// NeuroPLC ¡ª FourierKAN [28,16,4]
// C^2-BV Architecture: FourierKAN compiled via universal LUT extraction
// LUT points: 15, domain: [-3.0, 3.0]
// Proposition 9: M2 bounds guaranteed by C^2 property

FUNCTION_BLOCK "NeuroPLC_FourierKAN"
VAR_INPUT
    "feat_1" : REAL;
    "feat_2" : REAL;
    "feat_3" : REAL;
    "feat_4" : REAL;
    "feat_5" : REAL;
    "feat_6" : REAL;
    "feat_7" : REAL;
    "feat_8" : REAL;
    "feat_9" : REAL;
    "feat_10" : REAL;
    "feat_11" : REAL;
    "feat_12" : REAL;
    "feat_13" : REAL;
    "feat_14" : REAL;
    "feat_15" : REAL;
    "feat_16" : REAL;
    "feat_17" : REAL;
    "feat_18" : REAL;
    "feat_19" : REAL;
    "feat_20" : REAL;
    "feat_21" : REAL;
    "feat_22" : REAL;
    "feat_23" : REAL;
    "feat_24" : REAL;
    "feat_25" : REAL;
    "feat_26" : REAL;
    "feat_27" : REAL;
    "feat_28" : REAL;
    "trigger" : BOOL;
END_VAR

VAR_OUTPUT
    "class_output_1" : REAL;
    "class_output_2" : REAL;
    "class_output_3" : REAL;
    "class_output_4" : REAL;
    "max_confidence" : REAL;
    "predicted_class" : INT;
END_VAR

VAR
    "layer0_out_1" : REAL := 0.0;
    "layer0_out_2" : REAL := 0.0;
    "layer0_out_3" : REAL := 0.0;
    "layer0_out_4" : REAL := 0.0;
    "layer0_out_5" : REAL := 0.0;
    "layer0_out_6" : REAL := 0.0;
    "layer0_out_7" : REAL := 0.0;
    "layer0_out_8" : REAL := 0.0;
    "layer0_out_9" : REAL := 0.0;
    "layer0_out_10" : REAL := 0.0;
    "layer0_out_11" : REAL := 0.0;
    "layer0_out_12" : REAL := 0.0;
    "layer0_out_13" : REAL := 0.0;
    "layer0_out_14" : REAL := 0.0;
    "layer0_out_15" : REAL := 0.0;
    "layer0_out_16" : REAL := 0.0;
    "layer1_out_1" : REAL := 0.0;
    "layer1_out_2" : REAL := 0.0;
    "layer1_out_3" : REAL := 0.0;
    "layer1_out_4" : REAL := 0.0;
    "i" : INT;
    "k" : INT;
    "t" : REAL;
    "max_val" : REAL;
    "max_idx" : INT;
END_VAR

BEGIN
    IF NOT "trigger" THEN RETURN; END_IF;

    // === Layer 0 (28 -> 16) ===
    "layer0_out_1" := 0.0;
    // Edge (1->1): LUT interpolation
    "k" := 1;
    FOR "i" := 2 TO 15 DO
        IF "feat_1" >= -3.000000 AND "feat_1" <= 3.000000 THEN
    END_FOR;
    // Edge (2->1): LUT interpolation
    "k" := 1;
    FOR "i" := 2 TO 15 DO
    END_FOR;
    // Edge (3->1): LUT interpolation
    "k" := 1;
    FOR "i" := 2 TO 15 DO
    END_FOR;
    // Edge (4->1): LUT interpolation
    "k" := 1;
    FOR "i" := 2 TO 15 DO
    END_FOR;
    // Edge (5->1): LUT interpolation
    "k" := 1;
    FOR "i" := 2 TO 15 DO
    END_FOR;
    // Edge (6->1): LUT interpolation
    "k" := 1;
    FOR "i" := 2 TO 15 DO
    END_FOR;
    // Edge (7->1): LUT interpolation
    "k" := 1;
    FOR "i" := 2 TO 15 DO
    END_FOR;
    // Edge (8->1): LUT interpolation
    "k" := 1;
    FOR "i" := 2 TO 15 DO
    END_FOR;
    // Edge (9->1): LUT interpolation
    "k" := 1;
    FOR "i" := 2 TO 15 DO
    END_FOR;
    // Edge (10->1): LUT interpolation
    "k" := 1;
    FOR "i" := 2 TO 15 DO
    END_FOR;
    // Edge (11->1): LUT interpolation
    "k" := 1;
    FOR "i" := 2 TO 15 DO
    END_FOR;
    // Edge (12->1): LUT interpolation
    "k" := 1;
    FOR "i" := 2 TO 15 DO
    END_FOR;
    // Edge (13->1): LUT interpolation
    "k" := 1;
    FOR "i" := 2 TO 15 DO
    END_FOR;
    // Edge (14->1): LUT interpolation
    "k" := 1;
    FOR "i" := 2 TO 15 DO
    END_FOR;
    // Edge (15->1): LUT interpolation
    "k" := 1;
    FOR "i" := 2 TO 15 DO
    END_FOR;
    // Edge (16->1): LUT interpolation
    "k" := 1;
    FOR "i" := 2 TO 15 DO
    END_FOR;
    // Edge (17->1): LUT interpolation
    "k" := 1;
    FOR "i" := 2 TO 15 DO
    END_FOR;
    // Edge (18->1): LUT interpolation
    "k" := 1;
    FOR "i" := 2 TO 15 DO
    END_FOR;
    // Edge (19->1): LUT interpolation
    "k" := 1;
    FOR "i" := 2 TO 15 DO
    END_FOR;
    // Edge (20->1): LUT interpolation
    "k" := 1;
    FOR "i" := 2 TO 15 DO
    END_FOR;
    // Edge (21->1): LUT interpolation
    "k" := 1;
    FOR "i" := 2 TO 15 DO
    END_FOR;
    // Edge (22->1): LUT interpolation
    "k" := 1;
    FOR "i" := 2 TO 15 DO
    END_FOR;
    // Edge (23->1): LUT interpolation
    "k" := 1;
    FOR "i" := 2 TO 15 DO
    END_FOR;
    // Edge (24->1): LUT interpolation
    "k" := 1;
    FOR "i" := 2 TO 15 DO
    END_FOR;
    // Edge (25->1): LUT interpolation
    "k" := 1;
    FOR "i" := 2 TO 15 DO
    END_FOR;
    // Edge (26->1): LUT interpolation
    "k" := 1;
    FOR "i" := 2 TO 15 DO
    END_FOR;
    // Edge (27->1): LUT interpolation
    "k" := 1;
    FOR "i" := 2 TO 15 DO
    END_FOR;
    // Edge (28->1): LUT interpolation
    "k" := 1;
    FOR "i" := 2 TO 15 DO
    END_FOR;
    "layer0_out_2" := 0.0;
    // Edge (1->2): LUT interpolation
    "k" := 1;
    FOR "i" := 2 TO 15 DO
    END_FOR;
    // Edge (2->2): LUT interpolation
    "k" := 1;
    FOR "i" := 2 TO 15 DO
    END_FOR;
    // Edge (3->2): LUT interpolation
    "k" := 1;
    FOR "i" := 2 TO 15 DO
    END_FOR;
    // Edge (4->2): LUT interpolation
    "k" := 1;
    FOR "i" := 2 TO 15 DO
    END_FOR;
    // Edge (5->2): LUT interpolation
    "k" := 1;
    FOR "i" := 2 TO 15 DO
    END_FOR;
    // Edge (6->2): LUT interpolation
    "k" := 1;
    FOR "i" := 2 TO 15 DO
    END_FOR;
    // Edge (7->2): LUT interpolation
    "k" := 1;
    FOR "i" := 2 TO 15 DO
    END_FOR;
    // Edge (8->2): LUT interpolation
    "k" := 1;
    FOR "i" := 2 TO 15 DO
    END_FOR;
    // Edge (9->2): LUT interpolation
    "k" := 1;
    FOR "i" := 2 TO 15 DO
    END_FOR;
    // Edge (10->2): LUT interpolation
    "k" := 1;
    FOR "i" := 2 TO 15 DO
    END_FOR;
    // Edge (11->2): LUT interpolation
    "k" := 1;
    FOR "i" := 2 TO 15 DO
    END_FOR;
    // Edge (12->2): LUT interpolation
    "k" := 1;
    FOR "i" := 2 TO 15 DO
    END_FOR;
    // Edge (13->2): LUT interpolation
    "k" := 1;
    FOR "i" := 2 TO 15 DO
    END_FOR;
    // Edge (14->2): LUT interpolation
    "k" := 1;
    FOR "i" := 2 TO 15 DO
    END_FOR;
    // Edge (15->2): LUT interpolation
    "k" := 1;
    FOR "i" := 2 TO 15 DO
    END_FOR;
    // Edge (16->2): LUT interpolation
    "k" := 1;
    FOR "i" := 2 TO 15 DO
    END_FOR;
    // Edge (17->2): LUT interpolation
    "k" := 1;
    FOR "i" := 2 TO 15 DO
    END_FOR;
    // Edge (18->2): LUT interpolation
    "k" := 1;
    FOR "i" := 2 TO 15 DO
    END_FOR;
    // Edge (19->2): LUT interpolation
    "k" := 1;
    FOR "i" := 2 TO 15 DO
    END_FOR;
    // Edge (20->2): LUT interpolation
    "k" := 1;
    FOR "i" := 2 TO 15 DO
    END_FOR;
    // Edge (21->2): LUT interpolation
    "k" := 1;
    FOR "i" := 2 TO 15 DO
    END_FOR;
    // Edge (22->2): LUT interpolation
    "k" := 1;
    FOR "i" := 2 TO 15 DO
    END_FOR;
    // Edge (23->2): LUT interpolation
    "k" := 1;
    FOR "i" := 2 TO 15 DO
    END_FOR;
    // Edge (24->2): LUT interpolation
    "k" := 1;
    FOR "i" := 2 TO 15 DO
    END_FOR;
    // Edge (25->2): LUT interpolation
    "k" := 1;
    FOR "i" := 2 TO 15 DO
    END_FOR;
    // Edge (26->2): LUT interpolation
    "k" := 1;
    FOR "i" := 2 TO 15 DO
    END_FOR;
    // Edge (27->2): LUT interpolation
    "k" := 1;
    FOR "i" := 2 TO 15 DO
    END_FOR;
    // Edge (28->2): LUT interpolation
    "k" := 1;
    FOR "i" := 2 TO 15 DO
    END_FOR;
    "layer0_out_3" := 0.0;
    // Edge (1->3): LUT interpolation
    "k" := 1;
    FOR "i" := 2 TO 15 DO
    END_FOR;
    // Edge (2->3): LUT interpolation
    "k" := 1;
    FOR "i" := 2 TO 15 DO
    END_FOR;
    // Edge (3->3): LUT interpolation
    "k" := 1;
    FOR "i" := 2 TO 15 DO
    END_FOR;
    // Edge (4->3): LUT interpolation
    "k" := 1;
    FOR "i" := 2 TO 15 DO
    END_FOR;
    // Edge (5->3): LUT interpolation
    "k" := 1;
    FOR "i" := 2 TO 15 DO
    END_FOR;
    // Edge (6->3): LUT interpolation
    "k" := 1;
    FOR "i" := 2 TO 15 DO
    END_FOR;
    // Edge (7->3): LUT interpolation
    "k" := 1;
    FOR "i" := 2 TO 15 DO
    END_FOR;
    // Edge (8->3): LUT interpolation
    "k" := 1;
    FOR "i" := 2 TO 15 DO
    END_FOR;
    // Edge (9->3): LUT interpolation
    "k" := 1;
    FOR "i" := 2 TO 15 DO
    END_FOR;
    // Edge (10->3): LUT interpolation
    "k" := 1;
    FOR "i" := 2 TO 15 DO
    END_FOR;
    // Edge (11->3): LUT interpolation
    "k" := 1;
    FOR "i" := 2 TO 15 DO
    END_FOR;
    // Edge (12->3): LUT interpolation
    "k" := 1;
    FOR "i" := 2 TO 15 DO
    END_FOR;
    // Edge (13->3): LUT interpolation
    "k" := 1;
    FOR "i" := 2 TO 15 DO
    END_FOR;
    // Edge (14->3): LUT interpolation
    "k" := 1;
    FOR "i" := 2 TO 15 DO
    END_FOR;
    // Edge (15->3): LUT interpolation
    "k" := 1;
    FOR "i" := 2 TO 15 DO
    END_FOR;
    // Edge (16->3): LUT interpolation
    "k" := 1;
    FOR "i" := 2 TO 15 DO
    END_FOR;
    // Edge (17->3): LUT interpolation
    "k" := 1;
    FOR "i" := 2 TO 15 DO
    END_FOR;
    // Edge (18->3): LUT interpolation
    "k" := 1;
    FOR "i" := 2 TO 15 DO
    END_FOR;
    // Edge (19->3): LUT interpolation
    "k" := 1;
    FOR "i" := 2 TO 15 DO
    END_FOR;
    // Edge (20->3): LUT interpolation
    "k" := 1;
    FOR "i" := 2 TO 15 DO
    END_FOR;
    // Edge (21->3): LUT interpolation
    "k" := 1;
    FOR "i" := 2 TO 15 DO
    END_FOR;
    // Edge (22->3): LUT interpolation
    "k" := 1;
    FOR "i" := 2 TO 15 DO
    END_FOR;
    // Edge (23->3): LUT interpolation
    "k" := 1;
    FOR "i" := 2 TO 15 DO
    END_FOR;
    // Edge (24->3): LUT interpolation
    "k" := 1;
    FOR "i" := 2 TO 15 DO
    END_FOR;
    // Edge (25->3): LUT interpolation
    "k" := 1;
    FOR "i" := 2 TO 15 DO
    END_FOR;
    // Edge (26->3): LUT interpolation
    "k" := 1;
    FOR "i" := 2 TO 15 DO
    END_FOR;
    // Edge (27->3): LUT interpolation
    "k" := 1;
    FOR "i" := 2 TO 15 DO
    END_FOR;
    // Edge (28->3): LUT interpolation
    "k" := 1;
    FOR "i" := 2 TO 15 DO
    END_FOR;
    "layer0_out_4" := 0.0;
    // Edge (1->4): LUT interpolation
    "k" := 1;
    FOR "i" := 2 TO 15 DO
    END_FOR;
    // Edge (2->4): LUT interpolation
    "k" := 1;
    FOR "i" := 2 TO 15 DO
    END_FOR;
    // Edge (3->4): LUT interpolation
    "k" := 1;
    FOR "i" := 2 TO 15 DO
    END_FOR;
    // Edge (4->4): LUT interpolation
    "k" := 1;
    FOR "i" := 2 TO 15 DO
    END_FOR;
    // Edge (5->4): LUT interpolation
    "k" := 1;
    FOR "i" := 2 TO 15 DO
    END_FOR;
    // Edge (6->4): LUT interpolation
    "k" := 1;
    FOR "i" := 2 TO 15 DO
    END_FOR;
    // Edge (7->4): LUT interpolation
    "k" := 1;
    FOR "i" := 2 TO 15 DO
    END_FOR;
    // Edge (8->4): LUT interpolation
    "k" := 1;
    FOR "i" := 2 TO 15 DO
    END_FOR;
    // Edge (9->4): LUT interpolation
    "k" := 1;
    FOR "i" := 2 TO 15 DO
    END_FOR;
    // Edge (10->4): LUT interpolation
    "k" := 1;
    FOR "i" := 2 TO 15 DO
    END_FOR;
    // Edge (11->4): LUT interpolation
    "k" := 1;
    FOR "i" := 2 TO 15 DO
    END_FOR;
    // Edge (12->4): LUT interpolation
    "k" := 1;
    FOR "i" := 2 TO 15 DO
    END_FOR;
    // Edge (13->4): LUT interpolation
    "k" := 1;
    FOR "i" := 2 TO 15 DO
    END_FOR;
    // Edge (14->4): LUT interpolation
    "k" := 1;
    FOR "i" := 2 TO 15 DO
    END_FOR;
    // Edge (15->4): LUT interpolation
    "k" := 1;
    FOR "i" := 2 TO 15 DO
    END_FOR;
    // Edge (16->4): LUT interpolation
    "k" := 1;
    FOR "i" := 2 TO 15 DO
    END_FOR;
    // Edge (17->4): LUT interpolation
    "k" := 1;
    FOR "i" := 2 TO 15 DO
    END_FOR;
    // Edge (18->4): LUT interpolation
    "k" := 1;
    FOR "i" := 2 TO 15 DO
    END_FOR;
    // Edge (19->4): LUT interpolation
    "k" := 1;
    FOR "i" := 2 TO 15 DO
    END_FOR;
    // Edge (20->4): LUT interpolation
    "k" := 1;
    FOR "i" := 2 TO 15 DO
    END_FOR;
    // Edge (21->4): LUT interpolation
    "k" := 1;
    FOR "i" := 2 TO 15 DO
    END_FOR;
    // Edge (22->4): LUT interpolation
    "k" := 1;
    FOR "i" := 2 TO 15 DO
    END_FOR;
    // Edge (23->4): LUT interpolation
    "k" := 1;
    FOR "i" := 2 TO 15 DO
    END_FOR;
    // Edge (24->4): LUT interpolation
    "k" := 1;
    FOR "i" := 2 TO 15 DO
    END_FOR;
    // Edge (25->4): LUT interpolation
    "k" := 1;
    FOR "i" := 2 TO 15 DO
    END_FOR;
    // Edge (26->4): LUT interpolation
    "k" := 1;
    FOR "i" := 2 TO 15 DO
    END_FOR;
    // Edge (27->4): LUT interpolation
    "k" := 1;
    FOR "i" := 2 TO 15 DO
    END_FOR;
    // Edge (28->4): LUT interpolation
    "k" := 1;
    FOR "i" := 2 TO 15 DO
    END_FOR;
    "layer0_out_5" := 0.0;
    // Edge (1->5): LUT interpolation
    "k" := 1;
    FOR "i" := 2 TO 15 DO
    END_FOR;
    // Edge (2->5): LUT interpolation
    "k" := 1;
    FOR "i" := 2 TO 15 DO
    END_FOR;
    // Edge (3->5): LUT interpolation
    "k" := 1;
    FOR "i" := 2 TO 15 DO
    END_FOR;
    // Edge (4->5): LUT interpolation
    "k" := 1;
    FOR "i" := 2 TO 15 DO
    END_FOR;
    // Edge (5->5): LUT interpolation
    "k" := 1;
    FOR "i" := 2 TO 15 DO
    END_FOR;
    // Edge (6->5): LUT interpolation
    "k" := 1;
    FOR "i" := 2 TO 15 DO
    END_FOR;
    // Edge (7->5): LUT interpolation
    "k" := 1;
    FOR "i" := 2 TO 15 DO
    END_FOR;
    // Edge (8->5): LUT interpolation
    "k" := 1;
    FOR "i" := 2 TO 15 DO
    END_FOR;
    // Edge (9->5): LUT interpolation
    "k" := 1;
    FOR "i" := 2 TO 15 DO
    END_FOR;
    // Edge (10->5): LUT interpolation
    "k" := 1;
    FOR "i" := 2 TO 15 DO
    END_FOR;
    // Edge (11->5): LUT interpolation
    "k" := 1;
    FOR "i" := 2 TO 15 DO
    END_FOR;
    // Edge (12->5): LUT interpolation
    "k" := 1;
    FOR "i" := 2 TO 15 DO
    END_FOR;
    // Edge (13->5): LUT interpolation
    "k" := 1;
    FOR "i" := 2 TO 15 DO
    END_FOR;
    // Edge (14->5): LUT interpolation
    "k" := 1;
    FOR "i" := 2 TO 15 DO
    END_FOR;
    // Edge (15->5): LUT interpolation
    "k" := 1;
    FOR "i" := 2 TO 15 DO
    END_FOR;
    // Edge (16->5): LUT interpolation
    "k" := 1;
    FOR "i" := 2 TO 15 DO
    END_FOR;
    // Edge (17->5): LUT interpolation
    "k" := 1;
    FOR "i" := 2 TO 15 DO
    END_FOR;
    // Edge (18->5): LUT interpolation
    "k" := 1;
    FOR "i" := 2 TO 15 DO
    END_FOR;
    // Edge (19->5): LUT interpolation
    "k" := 1;
    FOR "i" := 2 TO 15 DO
    END_FOR;
    // Edge (20->5): LUT interpolation
    "k" := 1;
    FOR "i" := 2 TO 15 DO
    END_FOR;
    // Edge (21->5): LUT interpolation
    "k" := 1;
    FOR "i" := 2 TO 15 DO
    END_FOR;
    // Edge (22->5): LUT interpolation
    "k" := 1;
    FOR "i" := 2 TO 15 DO
    END_FOR;
    // Edge (23->5): LUT interpolation
    "k" := 1;
    FOR "i" := 2 TO 15 DO
    END_FOR;
    // Edge (24->5): LUT interpolation
    "k" := 1;
    FOR "i" := 2 TO 15 DO
    END_FOR;
    // Edge (25->5): LUT interpolation
    "k" := 1;
    FOR "i" := 2 TO 15 DO
    END_FOR;
    // Edge (26->5): LUT interpolation
    "k" := 1;
    FOR "i" := 2 TO 15 DO
    END_FOR;
    // Edge (27->5): LUT interpolation
    "k" := 1;
    FOR "i" := 2 TO 15 DO
    END_FOR;
    // Edge (28->5): LUT interpolation
    "k" := 1;
    FOR "i" := 2 TO 15 DO
    END_FOR;
    "layer0_out_6" := 0.0;
    // Edge (1->6): LUT interpolation
    "k" := 1;
    FOR "i" := 2 TO 15 DO
    END_FOR;
    // Edge (2->6): LUT interpolation
    "k" := 1;
    FOR "i" := 2 TO 15 DO
    END_FOR;
    // Edge (3->6): LUT interpolation
    "k" := 1;
    FOR "i" := 2 TO 15 DO
    END_FOR;
    // Edge (4->6): LUT interpolation
    "k" := 1;
    FOR "i" := 2 TO 15 DO
    END_FOR;
    // Edge (5->6): LUT interpolation
    "k" := 1;
    FOR "i" := 2 TO 15 DO
    END_FOR;
    // Edge (6->6): LUT interpolation
    "k" := 1;
    FOR "i" := 2 TO 15 DO
    END_FOR;
    // Edge (7->6): LUT interpolation
    "k" := 1;
    FOR "i" := 2 TO 15 DO
    END_FOR;
    // Edge (8->6): LUT interpolation
    "k" := 1;
    FOR "i" := 2 TO 15 DO
    END_FOR;
    // Edge (9->6): LUT interpolation
    "k" := 1;
    FOR "i" := 2 TO 15 DO
    END_FOR;
    // Edge (10->6): LUT interpolation
    "k" := 1;
    FOR "i" := 2 TO 15 DO
    END_FOR;
    // Edge (11->6): LUT interpolation
    "k" := 1;
    FOR "i" := 2 TO 15 DO
    END_FOR;
    // Edge (12->6): LUT interpolation
    "k" := 1;
    FOR "i" := 2 TO 15 DO
    END_FOR;
    // Edge (13->6): LUT interpolation
    "k" := 1;
    FOR "i" := 2 TO 15 DO
    END_FOR;
    // Edge (14->6): LUT interpolation
    "k" := 1;
    FOR "i" := 2 TO 15 DO
    END_FOR;
    // Edge (15->6): LUT interpolation
    "k" := 1;
    FOR "i" := 2 TO 15 DO
    END_FOR;
    // Edge (16->6): LUT interpolation
    "k" := 1;
    FOR "i" := 2 TO 15 DO
    END_FOR;
    // Edge (17->6): LUT interpolation
    "k" := 1;
    FOR "i" := 2 TO 15 DO
    END_FOR;
    // Edge (18->6): LUT interpolation
    "k" := 1;
    FOR "i" := 2 TO 15 DO
    END_FOR;
    // Edge (19->6): LUT interpolation
    "k" := 1;
    FOR "i" := 2 TO 15 DO
    END_FOR;
    // Edge (20->6): LUT interpolation
    "k" := 1;
    FOR "i" := 2 TO 15 DO
    END_FOR;
    // Edge (21->6): LUT interpolation
    "k" := 1;
    FOR "i" := 2 TO 15 DO
    END_FOR;
    // Edge (22->6): LUT interpolation
    "k" := 1;
    FOR "i" := 2 TO 15 DO
    END_FOR;
    // Edge (23->6): LUT interpolation
    "k" := 1;
    FOR "i" := 2 TO 15 DO
    END_FOR;
    // Edge (24->6): LUT interpolation
    "k" := 1;
    FOR "i" := 2 TO 15 DO
    END_FOR;
    // Edge (25->6): LUT interpolation
    "k" := 1;
    FOR "i" := 2 TO 15 DO
    END_FOR;
    // Edge (26->6): LUT interpolation
    "k" := 1;
    FOR "i" := 2 TO 15 DO
    END_FOR;
    // Edge (27->6): LUT interpolation
    "k" := 1;
    FOR "i" := 2 TO 15 DO
    END_FOR;
    // Edge (28->6): LUT interpolation
    "k" := 1;
    FOR "i" := 2 TO 15 DO
    END_FOR;
    "layer0_out_7" := 0.0;
    // Edge (1->7): LUT interpolation
    "k" := 1;
    FOR "i" := 2 TO 15 DO
    END_FOR;
    // Edge (2->7): LUT interpolation
    "k" := 1;
    FOR "i" := 2 TO 15 DO
    END_FOR;
    // Edge (3->7): LUT interpolation
    "k" := 1;
    FOR "i" := 2 TO 15 DO
    END_FOR;
    // Edge (4->7): LUT interpolation
    "k" := 1;
    FOR "i" := 2 TO 15 DO
    END_FOR;
    // Edge (5->7): LUT interpolation
    "k" := 1;
    FOR "i" := 2 TO 15 DO
    END_FOR;
    // Edge (6->7): LUT interpolation
    "k" := 1;
    FOR "i" := 2 TO 15 DO
    END_FOR;
    // Edge (7->7): LUT interpolation
    "k" := 1;
    FOR "i" := 2 TO 15 DO
    END_FOR;
    // Edge (8->7): LUT interpolation
    "k" := 1;
    FOR "i" := 2 TO 15 DO
    END_FOR;
    // Edge (9->7): LUT interpolation
    "k" := 1;
    FOR "i" := 2 TO 15 DO
    END_FOR;
    // Edge (10->7): LUT interpolation
    "k" := 1;
    FOR "i" := 2 TO 15 DO
    END_FOR;
    // Edge (11->7): LUT interpolation
    "k" := 1;
    FOR "i" := 2 TO 15 DO
    END_FOR;
    // Edge (12->7): LUT interpolation
    "k" := 1;
    FOR "i" := 2 TO 15 DO
    END_FOR;
    // Edge (13->7): LUT interpolation
    "k" := 1;
    FOR "i" := 2 TO 15 DO
    END_FOR;
    // Edge (14->7): LUT interpolation
    "k" := 1;
    FOR "i" := 2 TO 15 DO
    END_FOR;
    // Edge (15->7): LUT interpolation
    "k" := 1;
    FOR "i" := 2 TO 15 DO
    END_FOR;
    // Edge (16->7): LUT interpolation
    "k" := 1;
    FOR "i" := 2 TO 15 DO
    END_FOR;
    // Edge (17->7): LUT interpolation
    "k" := 1;
    FOR "i" := 2 TO 15 DO
    END_FOR;
    // Edge (18->7): LUT interpolation
    "k" := 1;
    FOR "i" := 2 TO 15 DO
    END_FOR;
    // Edge (19->7): LUT interpolation
    "k" := 1;
    FOR "i" := 2 TO 15 DO
    END_FOR;
    // Edge (20->7): LUT interpolation
    "k" := 1;
    FOR "i" := 2 TO 15 DO
    END_FOR;
    // Edge (21->7): LUT interpolation
    "k" := 1;
    FOR "i" := 2 TO 15 DO
    END_FOR;
    // Edge (22->7): LUT interpolation
    "k" := 1;
    FOR "i" := 2 TO 15 DO
    END_FOR;
    // Edge (23->7): LUT interpolation
    "k" := 1;
    FOR "i" := 2 TO 15 DO
    END_FOR;
    // Edge (24->7): LUT interpolation
    "k" := 1;
    FOR "i" := 2 TO 15 DO
    END_FOR;
    // Edge (25->7): LUT interpolation
    "k" := 1;
    FOR "i" := 2 TO 15 DO
    END_FOR;
    // Edge (26->7): LUT interpolation
    "k" := 1;
    FOR "i" := 2 TO 15 DO
    END_FOR;
    // Edge (27->7): LUT interpolation
    "k" := 1;
    FOR "i" := 2 TO 15 DO
    END_FOR;
    // Edge (28->7): LUT interpolation
    "k" := 1;
    FOR "i" := 2 TO 15 DO
    END_FOR;
    "layer0_out_8" := 0.0;
    // Edge (1->8): LUT interpolation
    "k" := 1;
    FOR "i" := 2 TO 15 DO
    END_FOR;
    // Edge (2->8): LUT interpolation
    "k" := 1;
    FOR "i" := 2 TO 15 DO
    END_FOR;
    // Edge (3->8): LUT interpolation
    "k" := 1;
    FOR "i" := 2 TO 15 DO
    END_FOR;
    // Edge (4->8): LUT interpolation
    "k" := 1;
    FOR "i" := 2 TO 15 DO
    END_FOR;
    // Edge (5->8): LUT interpolation
    "k" := 1;
    FOR "i" := 2 TO 15 DO
    END_FOR;
    // Edge (6->8): LUT interpolation
    "k" := 1;
    FOR "i" := 2 TO 15 DO
    END_FOR;
    // Edge (7->8): LUT interpolation
    "k" := 1;
    FOR "i" := 2 TO 15 DO
    END_FOR;
    // Edge (8->8): LUT interpolation
    "k" := 1;
    FOR "i" := 2 TO 15 DO
    END_FOR;
    // Edge (9->8): LUT interpolation
    "k" := 1;
    FOR "i" := 2 TO 15 DO
    END_FOR;
    // Edge (10->8): LUT interpolation
    "k" := 1;
    FOR "i" := 2 TO 15 DO
    END_FOR;
    // Edge (11->8): LUT interpolation
    "k" := 1;
    FOR "i" := 2 TO 15 DO
    END_FOR;
    // Edge (12->8): LUT interpolation
    "k" := 1;
    FOR "i" := 2 TO 15 DO
    END_FOR;
    // Edge (13->8): LUT interpolation
    "k" := 1;
    FOR "i" := 2 TO 15 DO
    END_FOR;
    // Edge (14->8): LUT interpolation
    "k" := 1;
    FOR "i" := 2 TO 15 DO
    END_FOR;
    // Edge (15->8): LUT interpolation
    "k" := 1;
    FOR "i" := 2 TO 15 DO
    END_FOR;
    // Edge (16->8): LUT interpolation
    "k" := 1;
    FOR "i" := 2 TO 15 DO
    END_FOR;
    // Edge (17->8): LUT interpolation
    "k" := 1;
    FOR "i" := 2 TO 15 DO
    END_FOR;
    // Edge (18->8): LUT interpolation
    "k" := 1;
    FOR "i" := 2 TO 15 DO
    END_FOR;
    // Edge (19->8): LUT interpolation
    "k" := 1;
    FOR "i" := 2 TO 15 DO
    END_FOR;
    // Edge (20->8): LUT interpolation
    "k" := 1;
    FOR "i" := 2 TO 15 DO
    END_FOR;
    // Edge (21->8): LUT interpolation
    "k" := 1;
    FOR "i" := 2 TO 15 DO
    END_FOR;
    // Edge (22->8): LUT interpolation
    "k" := 1;
    FOR "i" := 2 TO 15 DO
    END_FOR;
    // Edge (23->8): LUT interpolation
    "k" := 1;
    FOR "i" := 2 TO 15 DO
    END_FOR;
    // Edge (24->8): LUT interpolation
    "k" := 1;
    FOR "i" := 2 TO 15 DO
    END_FOR;
    // Edge (25->8): LUT interpolation
    "k" := 1;
    FOR "i" := 2 TO 15 DO
    END_FOR;
    // Edge (26->8): LUT interpolation
    "k" := 1;
    FOR "i" := 2 TO 15 DO
    END_FOR;
    // Edge (27->8): LUT interpolation
    "k" := 1;
    FOR "i" := 2 TO 15 DO
    END_FOR;
    // Edge (28->8): LUT interpolation
    "k" := 1;
    FOR "i" := 2 TO 15 DO
    END_FOR;
    "layer0_out_9" := 0.0;
    // Edge (1->9): LUT interpolation
    "k" := 1;
    FOR "i" := 2 TO 15 DO
    END_FOR;
    // Edge (2->9): LUT interpolation
    "k" := 1;
    FOR "i" := 2 TO 15 DO
    END_FOR;
    // Edge (3->9): LUT interpolation
    "k" := 1;
    FOR "i" := 2 TO 15 DO
    END_FOR;
    // Edge (4->9): LUT interpolation
    "k" := 1;
    FOR "i" := 2 TO 15 DO
    END_FOR;
    // Edge (5->9): LUT interpolation
    "k" := 1;
    FOR "i" := 2 TO 15 DO
    END_FOR;
    // Edge (6->9): LUT interpolation
    "k" := 1;
    FOR "i" := 2 TO 15 DO
    END_FOR;
    // Edge (7->9): LUT interpolation
    "k" := 1;
    FOR "i" := 2 TO 15 DO
    END_FOR;
    // Edge (8->9): LUT interpolation
    "k" := 1;
    FOR "i" := 2 TO 15 DO
    END_FOR;
    // Edge (9->9): LUT interpolation
    "k" := 1;
    FOR "i" := 2 TO 15 DO
    END_FOR;
    // Edge (10->9): LUT interpolation
    "k" := 1;
    FOR "i" := 2 TO 15 DO
    END_FOR;
    // Edge (11->9): LUT interpolation
    "k" := 1;
    FOR "i" := 2 TO 15 DO
    END_FOR;
    // Edge (12->9): LUT interpolation
    "k" := 1;
    FOR "i" := 2 TO 15 DO
    END_FOR;
    // Edge (13->9): LUT interpolation
    "k" := 1;
    FOR "i" := 2 TO 15 DO
    END_FOR;
    // Edge (14->9): LUT interpolation
    "k" := 1;
    FOR "i" := 2 TO 15 DO
    END_FOR;
    // Edge (15->9): LUT interpolation
    "k" := 1;
    FOR "i" := 2 TO 15 DO
    END_FOR;
    // Edge (16->9): LUT interpolation
    "k" := 1;
    FOR "i" := 2 TO 15 DO
    END_FOR;
    // Edge (17->9): LUT interpolation
    "k" := 1;
    FOR "i" := 2 TO 15 DO
    END_FOR;
    // Edge (18->9): LUT interpolation
    "k" := 1;
    FOR "i" := 2 TO 15 DO
    END_FOR;
    // Edge (19->9): LUT interpolation
    "k" := 1;
    FOR "i" := 2 TO 15 DO
    END_FOR;
    // Edge (20->9): LUT interpolation
    "k" := 1;
    FOR "i" := 2 TO 15 DO
    END_FOR;
    // Edge (21->9): LUT interpolation
    "k" := 1;
    FOR "i" := 2 TO 15 DO
    END_FOR;
    // Edge (22->9): LUT interpolation
    "k" := 1;
    FOR "i" := 2 TO 15 DO
    END_FOR;
    // Edge (23->9): LUT interpolation
    "k" := 1;
    FOR "i" := 2 TO 15 DO
    END_FOR;
    // Edge (24->9): LUT interpolation
    "k" := 1;
    FOR "i" := 2 TO 15 DO
    END_FOR;
    // Edge (25->9): LUT interpolation
    "k" := 1;
    FOR "i" := 2 TO 15 DO
    END_FOR;
    // Edge (26->9): LUT interpolation
    "k" := 1;
    FOR "i" := 2 TO 15 DO
    END_FOR;
    // Edge (27->9): LUT interpolation
    "k" := 1;
    FOR "i" := 2 TO 15 DO
    END_FOR;
    // Edge (28->9): LUT interpolation
    "k" := 1;
    FOR "i" := 2 TO 15 DO
    END_FOR;
    "layer0_out_10" := 0.0;
    // Edge (1->10): LUT interpolation
    "k" := 1;
    FOR "i" := 2 TO 15 DO
    END_FOR;
    // Edge (2->10): LUT interpolation
    "k" := 1;
    FOR "i" := 2 TO 15 DO
    END_FOR;
    // Edge (3->10): LUT interpolation
    "k" := 1;
    FOR "i" := 2 TO 15 DO
    END_FOR;
    // Edge (4->10): LUT interpolation
    "k" := 1;
    FOR "i" := 2 TO 15 DO
    END_FOR;
    // Edge (5->10): LUT interpolation
    "k" := 1;
    FOR "i" := 2 TO 15 DO
    END_FOR;
    // Edge (6->10): LUT interpolation
    "k" := 1;
    FOR "i" := 2 TO 15 DO
    END_FOR;
    // Edge (7->10): LUT interpolation
    "k" := 1;
    FOR "i" := 2 TO 15 DO
    END_FOR;
    // Edge (8->10): LUT interpolation
    "k" := 1;
    FOR "i" := 2 TO 15 DO
    END_FOR;
    // Edge (9->10): LUT interpolation
    "k" := 1;
    FOR "i" := 2 TO 15 DO
    END_FOR;
    // Edge (10->10): LUT interpolation
    "k" := 1;
    FOR "i" := 2 TO 15 DO
    END_FOR;
    // Edge (11->10): LUT interpolation
    "k" := 1;
    FOR "i" := 2 TO 15 DO
    END_FOR;
    // Edge (12->10): LUT interpolation
    "k" := 1;
    FOR "i" := 2 TO 15 DO
    END_FOR;
    // Edge (13->10): LUT interpolation
    "k" := 1;
    FOR "i" := 2 TO 15 DO
    END_FOR;
    // Edge (14->10): LUT interpolation
    "k" := 1;
    FOR "i" := 2 TO 15 DO
    END_FOR;
    // Edge (15->10): LUT interpolation
    "k" := 1;
    FOR "i" := 2 TO 15 DO
    END_FOR;
    // Edge (16->10): LUT interpolation
    "k" := 1;
    FOR "i" := 2 TO 15 DO
    END_FOR;
    // Edge (17->10): LUT interpolation
    "k" := 1;
    FOR "i" := 2 TO 15 DO
    END_FOR;
    // Edge (18->10): LUT interpolation
    "k" := 1;
    FOR "i" := 2 TO 15 DO
    END_FOR;
    // Edge (19->10): LUT interpolation
    "k" := 1;
    FOR "i" := 2 TO 15 DO
    END_FOR;
    // Edge (20->10): LUT interpolation
    "k" := 1;
    FOR "i" := 2 TO 15 DO
    END_FOR;
    // Edge (21->10): LUT interpolation
    "k" := 1;
    FOR "i" := 2 TO 15 DO
    END_FOR;
    // Edge (22->10): LUT interpolation
    "k" := 1;
    FOR "i" := 2 TO 15 DO
    END_FOR;
    // Edge (23->10): LUT interpolation
    "k" := 1;
    FOR "i" := 2 TO 15 DO
    END_FOR;
    // Edge (24->10): LUT interpolation
    "k" := 1;
    FOR "i" := 2 TO 15 DO
    END_FOR;
    // Edge (25->10): LUT interpolation
    "k" := 1;
    FOR "i" := 2 TO 15 DO
    END_FOR;
    // Edge (26->10): LUT interpolation
    "k" := 1;
    FOR "i" := 2 TO 15 DO
    END_FOR;
    // Edge (27->10): LUT interpolation
    "k" := 1;
    FOR "i" := 2 TO 15 DO
    END_FOR;
    // Edge (28->10): LUT interpolation
    "k" := 1;
    FOR "i" := 2 TO 15 DO
    END_FOR;
    "layer0_out_11" := 0.0;
    // Edge (1->11): LUT interpolation
    "k" := 1;
    FOR "i" := 2 TO 15 DO
    END_FOR;
    // Edge (2->11): LUT interpolation
    "k" := 1;
    FOR "i" := 2 TO 15 DO
    END_FOR;
    // Edge (3->11): LUT interpolation
    "k" := 1;
    FOR "i" := 2 TO 15 DO
    END_FOR;
    // Edge (4->11): LUT interpolation
    "k" := 1;
    FOR "i" := 2 TO 15 DO
    END_FOR;
    // Edge (5->11): LUT interpolation
    "k" := 1;
    FOR "i" := 2 TO 15 DO
    END_FOR;
    // Edge (6->11): LUT interpolation
    "k" := 1;
    FOR "i" := 2 TO 15 DO
    END_FOR;
    // Edge (7->11): LUT interpolation
    "k" := 1;
    FOR "i" := 2 TO 15 DO
    END_FOR;
    // Edge (8->11): LUT interpolation
    "k" := 1;
    FOR "i" := 2 TO 15 DO
    END_FOR;
    // Edge (9->11): LUT interpolation
    "k" := 1;
    FOR "i" := 2 TO 15 DO
    END_FOR;
    // Edge (10->11): LUT interpolation
    "k" := 1;
    FOR "i" := 2 TO 15 DO
    END_FOR;
    // Edge (11->11): LUT interpolation
    "k" := 1;
    FOR "i" := 2 TO 15 DO
    END_FOR;
    // Edge (12->11): LUT interpolation
    "k" := 1;
    FOR "i" := 2 TO 15 DO
    END_FOR;
    // Edge (13->11): LUT interpolation
    "k" := 1;
    FOR "i" := 2 TO 15 DO
    END_FOR;
    // Edge (14->11): LUT interpolation
    "k" := 1;
    FOR "i" := 2 TO 15 DO
    END_FOR;
    // Edge (15->11): LUT interpolation
    "k" := 1;
    FOR "i" := 2 TO 15 DO
    END_FOR;
    // Edge (16->11): LUT interpolation
    "k" := 1;
    FOR "i" := 2 TO 15 DO
    END_FOR;
    // Edge (17->11): LUT interpolation
    "k" := 1;
    FOR "i" := 2 TO 15 DO
    END_FOR;
    // Edge (18->11): LUT interpolation
    "k" := 1;
    FOR "i" := 2 TO 15 DO
    END_FOR;
    // Edge (19->11): LUT interpolation
    "k" := 1;
    FOR "i" := 2 TO 15 DO
    END_FOR;
    // Edge (20->11): LUT interpolation
    "k" := 1;
    FOR "i" := 2 TO 15 DO
    END_FOR;
    // Edge (21->11): LUT interpolation
    "k" := 1;
    FOR "i" := 2 TO 15 DO
    END_FOR;
    // Edge (22->11): LUT interpolation
    "k" := 1;
    FOR "i" := 2 TO 15 DO
    END_FOR;
    // Edge (23->11): LUT interpolation
    "k" := 1;
    FOR "i" := 2 TO 15 DO
    END_FOR;
    // Edge (24->11): LUT interpolation
    "k" := 1;
    FOR "i" := 2 TO 15 DO
    END_FOR;
    // Edge (25->11): LUT interpolation
    "k" := 1;
    FOR "i" := 2 TO 15 DO
    END_FOR;
    // Edge (26->11): LUT interpolation
    "k" := 1;
    FOR "i" := 2 TO 15 DO
    END_FOR;
    // Edge (27->11): LUT interpolation
    "k" := 1;
    FOR "i" := 2 TO 15 DO
    END_FOR;
    // Edge (28->11): LUT interpolation
    "k" := 1;
    FOR "i" := 2 TO 15 DO
    END_FOR;
    "layer0_out_12" := 0.0;
    // Edge (1->12): LUT interpolation
    "k" := 1;
    FOR "i" := 2 TO 15 DO
    END_FOR;
    // Edge (2->12): LUT interpolation
    "k" := 1;
    FOR "i" := 2 TO 15 DO
    END_FOR;
    // Edge (3->12): LUT interpolation
    "k" := 1;
    FOR "i" := 2 TO 15 DO
    END_FOR;
    // Edge (4->12): LUT interpolation
    "k" := 1;
    FOR "i" := 2 TO 15 DO
    END_FOR;
    // Edge (5->12): LUT interpolation
    "k" := 1;
    FOR "i" := 2 TO 15 DO
    END_FOR;
    // Edge (6->12): LUT interpolation
    "k" := 1;
    FOR "i" := 2 TO 15 DO
    END_FOR;
    // Edge (7->12): LUT interpolation
    "k" := 1;
    FOR "i" := 2 TO 15 DO
    END_FOR;
    // Edge (8->12): LUT interpolation
    "k" := 1;
    FOR "i" := 2 TO 15 DO
    END_FOR;
    // Edge (9->12): LUT interpolation
    "k" := 1;
    FOR "i" := 2 TO 15 DO
    END_FOR;
    // Edge (10->12): LUT interpolation
    "k" := 1;
    FOR "i" := 2 TO 15 DO
    END_FOR;
    // Edge (11->12): LUT interpolation
    "k" := 1;
    FOR "i" := 2 TO 15 DO
    END_FOR;
    // Edge (12->12): LUT interpolation
    "k" := 1;
    FOR "i" := 2 TO 15 DO
    END_FOR;
    // Edge (13->12): LUT interpolation
    "k" := 1;
    FOR "i" := 2 TO 15 DO
    END_FOR;
    // Edge (14->12): LUT interpolation
    "k" := 1;
    FOR "i" := 2 TO 15 DO
    END_FOR;
    // Edge (15->12): LUT interpolation
    "k" := 1;
    FOR "i" := 2 TO 15 DO
    END_FOR;
    // Edge (16->12): LUT interpolation
    "k" := 1;
    FOR "i" := 2 TO 15 DO
    END_FOR;
    // Edge (17->12): LUT interpolation
    "k" := 1;
    FOR "i" := 2 TO 15 DO
    END_FOR;
    // Edge (18->12): LUT interpolation
    "k" := 1;
    FOR "i" := 2 TO 15 DO
    END_FOR;
    // Edge (19->12): LUT interpolation
    "k" := 1;
    FOR "i" := 2 TO 15 DO
    END_FOR;
    // Edge (20->12): LUT interpolation
    "k" := 1;
    FOR "i" := 2 TO 15 DO
    END_FOR;
    // Edge (21->12): LUT interpolation
    "k" := 1;
    FOR "i" := 2 TO 15 DO
    END_FOR;
    // Edge (22->12): LUT interpolation
    "k" := 1;
    FOR "i" := 2 TO 15 DO
    END_FOR;
    // Edge (23->12): LUT interpolation
    "k" := 1;
    FOR "i" := 2 TO 15 DO
    END_FOR;
    // Edge (24->12): LUT interpolation
    "k" := 1;
    FOR "i" := 2 TO 15 DO
    END_FOR;
    // Edge (25->12): LUT interpolation
    "k" := 1;
    FOR "i" := 2 TO 15 DO
    END_FOR;
    // Edge (26->12): LUT interpolation
    "k" := 1;
    FOR "i" := 2 TO 15 DO
    END_FOR;
    // Edge (27->12): LUT interpolation
    "k" := 1;
    FOR "i" := 2 TO 15 DO
    END_FOR;
    // Edge (28->12): LUT interpolation
    "k" := 1;
    FOR "i" := 2 TO 15 DO
    END_FOR;
    "layer0_out_13" := 0.0;
    // Edge (1->13): LUT interpolation
    "k" := 1;
    FOR "i" := 2 TO 15 DO
    END_FOR;
    // Edge (2->13): LUT interpolation
    "k" := 1;
    FOR "i" := 2 TO 15 DO
    END_FOR;
    // Edge (3->13): LUT interpolation
    "k" := 1;
    FOR "i" := 2 TO 15 DO
    END_FOR;
    // Edge (4->13): LUT interpolation
    "k" := 1;
    FOR "i" := 2 TO 15 DO
    END_FOR;
    // Edge (5->13): LUT interpolation
    "k" := 1;
    FOR "i" := 2 TO 15 DO
    END_FOR;
    // Edge (6->13): LUT interpolation
    "k" := 1;
    FOR "i" := 2 TO 15 DO
    END_FOR;
    // Edge (7->13): LUT interpolation
    "k" := 1;
    FOR "i" := 2 TO 15 DO
    END_FOR;
    // Edge (8->13): LUT interpolation
    "k" := 1;
    FOR "i" := 2 TO 15 DO
    END_FOR;
    // Edge (9->13): LUT interpolation
    "k" := 1;
    FOR "i" := 2 TO 15 DO
    END_FOR;
    // Edge (10->13): LUT interpolation
    "k" := 1;
    FOR "i" := 2 TO 15 DO
    END_FOR;
    // Edge (11->13): LUT interpolation
    "k" := 1;
    FOR "i" := 2 TO 15 DO
    END_FOR;
    // Edge (12->13): LUT interpolation
    "k" := 1;
    FOR "i" := 2 TO 15 DO
    END_FOR;
    // Edge (13->13): LUT interpolation
    "k" := 1;
    FOR "i" := 2 TO 15 DO
    END_FOR;
    // Edge (14->13): LUT interpolation
    "k" := 1;
    FOR "i" := 2 TO 15 DO
    END_FOR;
    // Edge (15->13): LUT interpolation
    "k" := 1;
    FOR "i" := 2 TO 15 DO
    END_FOR;
    // Edge (16->13): LUT interpolation
    "k" := 1;
    FOR "i" := 2 TO 15 DO
    END_FOR;
    // Edge (17->13): LUT interpolation
    "k" := 1;
    FOR "i" := 2 TO 15 DO
    END_FOR;
    // Edge (18->13): LUT interpolation
    "k" := 1;
    FOR "i" := 2 TO 15 DO
    END_FOR;
    // Edge (19->13): LUT interpolation
    "k" := 1;
    FOR "i" := 2 TO 15 DO
    END_FOR;
    // Edge (20->13): LUT interpolation
    "k" := 1;
    FOR "i" := 2 TO 15 DO
    END_FOR;
    // Edge (21->13): LUT interpolation
    "k" := 1;
    FOR "i" := 2 TO 15 DO
    END_FOR;
    // Edge (22->13): LUT interpolation
    "k" := 1;
    FOR "i" := 2 TO 15 DO
    END_FOR;
    // Edge (23->13): LUT interpolation
    "k" := 1;
    FOR "i" := 2 TO 15 DO
    END_FOR;
    // Edge (24->13): LUT interpolation
    "k" := 1;
    FOR "i" := 2 TO 15 DO
    END_FOR;
    // Edge (25->13): LUT interpolation
    "k" := 1;
    FOR "i" := 2 TO 15 DO
    END_FOR;
    // Edge (26->13): LUT interpolation
    "k" := 1;
    FOR "i" := 2 TO 15 DO
    END_FOR;
    // Edge (27->13): LUT interpolation
    "k" := 1;
    FOR "i" := 2 TO 15 DO
    END_FOR;
    // Edge (28->13): LUT interpolation
    "k" := 1;
    FOR "i" := 2 TO 15 DO
    END_FOR;
    "layer0_out_14" := 0.0;
    // Edge (1->14): LUT interpolation
    "k" := 1;
    FOR "i" := 2 TO 15 DO
    END_FOR;
    // Edge (2->14): LUT interpolation
    "k" := 1;
    FOR "i" := 2 TO 15 DO
    END_FOR;
    // Edge (3->14): LUT interpolation
    "k" := 1;
    FOR "i" := 2 TO 15 DO
    END_FOR;
    // Edge (4->14): LUT interpolation
    "k" := 1;
    FOR "i" := 2 TO 15 DO
    END_FOR;
    // Edge (5->14): LUT interpolation
    "k" := 1;
    FOR "i" := 2 TO 15 DO
    END_FOR;
    // Edge (6->14): LUT interpolation
    "k" := 1;
    FOR "i" := 2 TO 15 DO
    END_FOR;
    // Edge (7->14): LUT interpolation
    "k" := 1;
    FOR "i" := 2 TO 15 DO
    END_FOR;
    // Edge (8->14): LUT interpolation
    "k" := 1;
    FOR "i" := 2 TO 15 DO
    END_FOR;
    // Edge (9->14): LUT interpolation
    "k" := 1;
    FOR "i" := 2 TO 15 DO
    END_FOR;
    // Edge (10->14): LUT interpolation
    "k" := 1;
    FOR "i" := 2 TO 15 DO
    END_FOR;
    // Edge (11->14): LUT interpolation
    "k" := 1;
    FOR "i" := 2 TO 15 DO
    END_FOR;
    // Edge (12->14): LUT interpolation
    "k" := 1;
    FOR "i" := 2 TO 15 DO
    END_FOR;
    // Edge (13->14): LUT interpolation
    "k" := 1;
    FOR "i" := 2 TO 15 DO
    END_FOR;
    // Edge (14->14): LUT interpolation
    "k" := 1;
    FOR "i" := 2 TO 15 DO
    END_FOR;
    // Edge (15->14): LUT interpolation
    "k" := 1;
    FOR "i" := 2 TO 15 DO
    END_FOR;
    // Edge (16->14): LUT interpolation
    "k" := 1;
    FOR "i" := 2 TO 15 DO
    END_FOR;
    // Edge (17->14): LUT interpolation
    "k" := 1;
    FOR "i" := 2 TO 15 DO
    END_FOR;
    // Edge (18->14): LUT interpolation
    "k" := 1;
    FOR "i" := 2 TO 15 DO
    END_FOR;
    // Edge (19->14): LUT interpolation
    "k" := 1;
    FOR "i" := 2 TO 15 DO
    END_FOR;
    // Edge (20->14): LUT interpolation
    "k" := 1;
    FOR "i" := 2 TO 15 DO
    END_FOR;
    // Edge (21->14): LUT interpolation
    "k" := 1;
    FOR "i" := 2 TO 15 DO
    END_FOR;
    // Edge (22->14): LUT interpolation
    "k" := 1;
    FOR "i" := 2 TO 15 DO
    END_FOR;
    // Edge (23->14): LUT interpolation
    "k" := 1;
    FOR "i" := 2 TO 15 DO
    END_FOR;
    // Edge (24->14): LUT interpolation
    "k" := 1;
    FOR "i" := 2 TO 15 DO
    END_FOR;
    // Edge (25->14): LUT interpolation
    "k" := 1;
    FOR "i" := 2 TO 15 DO
    END_FOR;
    // Edge (26->14): LUT interpolation
    "k" := 1;
    FOR "i" := 2 TO 15 DO
    END_FOR;
    // Edge (27->14): LUT interpolation
    "k" := 1;
    FOR "i" := 2 TO 15 DO
    END_FOR;
    // Edge (28->14): LUT interpolation
    "k" := 1;
    FOR "i" := 2 TO 15 DO
    END_FOR;
    "layer0_out_15" := 0.0;
    // Edge (1->15): LUT interpolation
    "k" := 1;
    FOR "i" := 2 TO 15 DO
    END_FOR;
    // Edge (2->15): LUT interpolation
    "k" := 1;
    FOR "i" := 2 TO 15 DO
    END_FOR;
    // Edge (3->15): LUT interpolation
    "k" := 1;
    FOR "i" := 2 TO 15 DO
    END_FOR;
    // Edge (4->15): LUT interpolation
    "k" := 1;
    FOR "i" := 2 TO 15 DO
    END_FOR;
    // Edge (5->15): LUT interpolation
    "k" := 1;
    FOR "i" := 2 TO 15 DO
    END_FOR;
    // Edge (6->15): LUT interpolation
    "k" := 1;
    FOR "i" := 2 TO 15 DO
    END_FOR;
    // Edge (7->15): LUT interpolation
    "k" := 1;
    FOR "i" := 2 TO 15 DO
    END_FOR;
    // Edge (8->15): LUT interpolation
    "k" := 1;
    FOR "i" := 2 TO 15 DO
    END_FOR;
    // Edge (9->15): LUT interpolation
    "k" := 1;
    FOR "i" := 2 TO 15 DO
    END_FOR;
    // Edge (10->15): LUT interpolation
    "k" := 1;
    FOR "i" := 2 TO 15 DO
    END_FOR;
    // Edge (11->15): LUT interpolation
    "k" := 1;
    FOR "i" := 2 TO 15 DO
    END_FOR;
    // Edge (12->15): LUT interpolation
    "k" := 1;
    FOR "i" := 2 TO 15 DO
    END_FOR;
    // Edge (13->15): LUT interpolation
    "k" := 1;
    FOR "i" := 2 TO 15 DO
    END_FOR;
    // Edge (14->15): LUT interpolation
    "k" := 1;
    FOR "i" := 2 TO 15 DO
    END_FOR;
    // Edge (15->15): LUT interpolation
    "k" := 1;
    FOR "i" := 2 TO 15 DO
    END_FOR;
    // Edge (16->15): LUT interpolation
    "k" := 1;
    FOR "i" := 2 TO 15 DO
    END_FOR;
    // Edge (17->15): LUT interpolation
    "k" := 1;
    FOR "i" := 2 TO 15 DO
    END_FOR;
    // Edge (18->15): LUT interpolation
    "k" := 1;
    FOR "i" := 2 TO 15 DO
    END_FOR;
    // Edge (19->15): LUT interpolation
    "k" := 1;
    FOR "i" := 2 TO 15 DO
    END_FOR;
    // Edge (20->15): LUT interpolation
    "k" := 1;
    FOR "i" := 2 TO 15 DO
    END_FOR;
    // Edge (21->15): LUT interpolation
    "k" := 1;
    FOR "i" := 2 TO 15 DO
    END_FOR;
    // Edge (22->15): LUT interpolation
    "k" := 1;
    FOR "i" := 2 TO 15 DO
    END_FOR;
    // Edge (23->15): LUT interpolation
    "k" := 1;
    FOR "i" := 2 TO 15 DO
    END_FOR;
    // Edge (24->15): LUT interpolation
    "k" := 1;
    FOR "i" := 2 TO 15 DO
    END_FOR;
    // Edge (25->15): LUT interpolation
    "k" := 1;
    FOR "i" := 2 TO 15 DO
    END_FOR;
    // Edge (26->15): LUT interpolation
    "k" := 1;
    FOR "i" := 2 TO 15 DO
    END_FOR;
    // Edge (27->15): LUT interpolation
    "k" := 1;
    FOR "i" := 2 TO 15 DO
    END_FOR;
    // Edge (28->15): LUT interpolation
    "k" := 1;
    FOR "i" := 2 TO 15 DO
    END_FOR;
    "layer0_out_16" := 0.0;
    // Edge (1->16): LUT interpolation
    "k" := 1;
    FOR "i" := 2 TO 15 DO
    END_FOR;
    // Edge (2->16): LUT interpolation
    "k" := 1;
    FOR "i" := 2 TO 15 DO
    END_FOR;
    // Edge (3->16): LUT interpolation
    "k" := 1;
    FOR "i" := 2 TO 15 DO
    END_FOR;
    // Edge (4->16): LUT interpolation
    "k" := 1;
    FOR "i" := 2 TO 15 DO
    END_FOR;
    // Edge (5->16): LUT interpolation
    "k" := 1;
    FOR "i" := 2 TO 15 DO
    END_FOR;
    // Edge (6->16): LUT interpolation
    "k" := 1;
    FOR "i" := 2 TO 15 DO
    END_FOR;
    // Edge (7->16): LUT interpolation
    "k" := 1;
    FOR "i" := 2 TO 15 DO
    END_FOR;
    // Edge (8->16): LUT interpolation
    "k" := 1;
    FOR "i" := 2 TO 15 DO
    END_FOR;
    // Edge (9->16): LUT interpolation
    "k" := 1;
    FOR "i" := 2 TO 15 DO
    END_FOR;
    // Edge (10->16): LUT interpolation
    "k" := 1;
    FOR "i" := 2 TO 15 DO
    END_FOR;
    // Edge (11->16): LUT interpolation
    "k" := 1;
    FOR "i" := 2 TO 15 DO
    END_FOR;
    // Edge (12->16): LUT interpolation
    "k" := 1;
    FOR "i" := 2 TO 15 DO
    END_FOR;
    // Edge (13->16): LUT interpolation
    "k" := 1;
    FOR "i" := 2 TO 15 DO
    END_FOR;
    // Edge (14->16): LUT interpolation
    "k" := 1;
    FOR "i" := 2 TO 15 DO
    END_FOR;
    // Edge (15->16): LUT interpolation
    "k" := 1;
    FOR "i" := 2 TO 15 DO
    END_FOR;
    // Edge (16->16): LUT interpolation
    "k" := 1;
    FOR "i" := 2 TO 15 DO
    END_FOR;
    // Edge (17->16): LUT interpolation
    "k" := 1;
    FOR "i" := 2 TO 15 DO
    END_FOR;
    // Edge (18->16): LUT interpolation
    "k" := 1;
    FOR "i" := 2 TO 15 DO
    END_FOR;
    // Edge (19->16): LUT interpolation
    "k" := 1;
    FOR "i" := 2 TO 15 DO
    END_FOR;
    // Edge (20->16): LUT interpolation
    "k" := 1;
    FOR "i" := 2 TO 15 DO
    END_FOR;
    // Edge (21->16): LUT interpolation
    "k" := 1;
    FOR "i" := 2 TO 15 DO
    END_FOR;
    // Edge (22->16): LUT interpolation
    "k" := 1;
    FOR "i" := 2 TO 15 DO
    END_FOR;
    // Edge (23->16): LUT interpolation
    "k" := 1;
    FOR "i" := 2 TO 15 DO
    END_FOR;
    // Edge (24->16): LUT interpolation
    "k" := 1;
    FOR "i" := 2 TO 15 DO
    END_FOR;
    // Edge (25->16): LUT interpolation
    "k" := 1;
    FOR "i" := 2 TO 15 DO
    END_FOR;
    // Edge (26->16): LUT interpolation
    "k" := 1;
    FOR "i" := 2 TO 15 DO
    END_FOR;
    // Edge (27->16): LUT interpolation
    "k" := 1;
    FOR "i" := 2 TO 15 DO
    END_FOR;
    // Edge (28->16): LUT interpolation
    "k" := 1;
    FOR "i" := 2 TO 15 DO
    END_FOR;

    // === Layer 1 (16 -> 4) ===
    "layer1_out_1" := 0.0;
    // Edge (1->1): LUT interpolation
    "k" := 1;
    FOR "i" := 2 TO 15 DO
        IF "feat_1" >= -3.000000 AND "feat_1" <= 3.000000 THEN
    END_FOR;
    // Edge (2->1): LUT interpolation
    "k" := 1;
    FOR "i" := 2 TO 15 DO
    END_FOR;
    // Edge (3->1): LUT interpolation
    "k" := 1;
    FOR "i" := 2 TO 15 DO
    END_FOR;
    // Edge (4->1): LUT interpolation
    "k" := 1;
    FOR "i" := 2 TO 15 DO
    END_FOR;
    // Edge (5->1): LUT interpolation
    "k" := 1;
    FOR "i" := 2 TO 15 DO
    END_FOR;
    // Edge (6->1): LUT interpolation
    "k" := 1;
    FOR "i" := 2 TO 15 DO
    END_FOR;
    // Edge (7->1): LUT interpolation
    "k" := 1;
    FOR "i" := 2 TO 15 DO
    END_FOR;
    // Edge (8->1): LUT interpolation
    "k" := 1;
    FOR "i" := 2 TO 15 DO
    END_FOR;
    // Edge (9->1): LUT interpolation
    "k" := 1;
    FOR "i" := 2 TO 15 DO
    END_FOR;
    // Edge (10->1): LUT interpolation
    "k" := 1;
    FOR "i" := 2 TO 15 DO
    END_FOR;
    // Edge (11->1): LUT interpolation
    "k" := 1;
    FOR "i" := 2 TO 15 DO
    END_FOR;
    // Edge (12->1): LUT interpolation
    "k" := 1;
    FOR "i" := 2 TO 15 DO
    END_FOR;
    // Edge (13->1): LUT interpolation
    "k" := 1;
    FOR "i" := 2 TO 15 DO
    END_FOR;
    // Edge (14->1): LUT interpolation
    "k" := 1;
    FOR "i" := 2 TO 15 DO
    END_FOR;
    // Edge (15->1): LUT interpolation
    "k" := 1;
    FOR "i" := 2 TO 15 DO
    END_FOR;
    // Edge (16->1): LUT interpolation
    "k" := 1;
    FOR "i" := 2 TO 15 DO
    END_FOR;
    "layer1_out_2" := 0.0;
    // Edge (1->2): LUT interpolation
    "k" := 1;
    FOR "i" := 2 TO 15 DO
    END_FOR;
    // Edge (2->2): LUT interpolation
    "k" := 1;
    FOR "i" := 2 TO 15 DO
    END_FOR;
    // Edge (3->2): LUT interpolation
    "k" := 1;
    FOR "i" := 2 TO 15 DO
    END_FOR;
    // Edge (4->2): LUT interpolation
    "k" := 1;
    FOR "i" := 2 TO 15 DO
    END_FOR;
    // Edge (5->2): LUT interpolation
    "k" := 1;
    FOR "i" := 2 TO 15 DO
    END_FOR;
    // Edge (6->2): LUT interpolation
    "k" := 1;
    FOR "i" := 2 TO 15 DO
    END_FOR;
    // Edge (7->2): LUT interpolation
    "k" := 1;
    FOR "i" := 2 TO 15 DO
    END_FOR;
    // Edge (8->2): LUT interpolation
    "k" := 1;
    FOR "i" := 2 TO 15 DO
    END_FOR;
    // Edge (9->2): LUT interpolation
    "k" := 1;
    FOR "i" := 2 TO 15 DO
    END_FOR;
    // Edge (10->2): LUT interpolation
    "k" := 1;
    FOR "i" := 2 TO 15 DO
    END_FOR;
    // Edge (11->2): LUT interpolation
    "k" := 1;
    FOR "i" := 2 TO 15 DO
    END_FOR;
    // Edge (12->2): LUT interpolation
    "k" := 1;
    FOR "i" := 2 TO 15 DO
    END_FOR;
    // Edge (13->2): LUT interpolation
    "k" := 1;
    FOR "i" := 2 TO 15 DO
    END_FOR;
    // Edge (14->2): LUT interpolation
    "k" := 1;
    FOR "i" := 2 TO 15 DO
    END_FOR;
    // Edge (15->2): LUT interpolation
    "k" := 1;
    FOR "i" := 2 TO 15 DO
    END_FOR;
    // Edge (16->2): LUT interpolation
    "k" := 1;
    FOR "i" := 2 TO 15 DO
    END_FOR;
    "layer1_out_3" := 0.0;
    // Edge (1->3): LUT interpolation
    "k" := 1;
    FOR "i" := 2 TO 15 DO
    END_FOR;
    // Edge (2->3): LUT interpolation
    "k" := 1;
    FOR "i" := 2 TO 15 DO
    END_FOR;
    // Edge (3->3): LUT interpolation
    "k" := 1;
    FOR "i" := 2 TO 15 DO
    END_FOR;
    // Edge (4->3): LUT interpolation
    "k" := 1;
    FOR "i" := 2 TO 15 DO
    END_FOR;
    // Edge (5->3): LUT interpolation
    "k" := 1;
    FOR "i" := 2 TO 15 DO
    END_FOR;
    // Edge (6->3): LUT interpolation
    "k" := 1;
    FOR "i" := 2 TO 15 DO
    END_FOR;
    // Edge (7->3): LUT interpolation
    "k" := 1;
    FOR "i" := 2 TO 15 DO
    END_FOR;
    // Edge (8->3): LUT interpolation
    "k" := 1;
    FOR "i" := 2 TO 15 DO
    END_FOR;
    // Edge (9->3): LUT interpolation
    "k" := 1;
    FOR "i" := 2 TO 15 DO
    END_FOR;
    // Edge (10->3): LUT interpolation
    "k" := 1;
    FOR "i" := 2 TO 15 DO
    END_FOR;
    // Edge (11->3): LUT interpolation
    "k" := 1;
    FOR "i" := 2 TO 15 DO
    END_FOR;
    // Edge (12->3): LUT interpolation
    "k" := 1;
    FOR "i" := 2 TO 15 DO
    END_FOR;
    // Edge (13->3): LUT interpolation
    "k" := 1;
    FOR "i" := 2 TO 15 DO
    END_FOR;
    // Edge (14->3): LUT interpolation
    "k" := 1;
    FOR "i" := 2 TO 15 DO
    END_FOR;
    // Edge (15->3): LUT interpolation
    "k" := 1;
    FOR "i" := 2 TO 15 DO
    END_FOR;
    // Edge (16->3): LUT interpolation
    "k" := 1;
    FOR "i" := 2 TO 15 DO
    END_FOR;
    "layer1_out_4" := 0.0;
    // Edge (1->4): LUT interpolation
    "k" := 1;
    FOR "i" := 2 TO 15 DO
    END_FOR;
    // Edge (2->4): LUT interpolation
    "k" := 1;
    FOR "i" := 2 TO 15 DO
    END_FOR;
    // Edge (3->4): LUT interpolation
    "k" := 1;
    FOR "i" := 2 TO 15 DO
    END_FOR;
    // Edge (4->4): LUT interpolation
    "k" := 1;
    FOR "i" := 2 TO 15 DO
    END_FOR;
    // Edge (5->4): LUT interpolation
    "k" := 1;
    FOR "i" := 2 TO 15 DO
    END_FOR;
    // Edge (6->4): LUT interpolation
    "k" := 1;
    FOR "i" := 2 TO 15 DO
    END_FOR;
    // Edge (7->4): LUT interpolation
    "k" := 1;
    FOR "i" := 2 TO 15 DO
    END_FOR;
    // Edge (8->4): LUT interpolation
    "k" := 1;
    FOR "i" := 2 TO 15 DO
    END_FOR;
    // Edge (9->4): LUT interpolation
    "k" := 1;
    FOR "i" := 2 TO 15 DO
    END_FOR;
    // Edge (10->4): LUT interpolation
    "k" := 1;
    FOR "i" := 2 TO 15 DO
    END_FOR;
    // Edge (11->4): LUT interpolation
    "k" := 1;
    FOR "i" := 2 TO 15 DO
    END_FOR;
    // Edge (12->4): LUT interpolation
    "k" := 1;
    FOR "i" := 2 TO 15 DO
    END_FOR;
    // Edge (13->4): LUT interpolation
    "k" := 1;
    FOR "i" := 2 TO 15 DO
    END_FOR;
    // Edge (14->4): LUT interpolation
    "k" := 1;
    FOR "i" := 2 TO 15 DO
    END_FOR;
    // Edge (15->4): LUT interpolation
    "k" := 1;
    FOR "i" := 2 TO 15 DO
    END_FOR;
    // Edge (16->4): LUT interpolation
    "k" := 1;
    FOR "i" := 2 TO 15 DO
    END_FOR;

    // === Softmax ===
    "max_val" := "layer1_out_1";
    IF "layer1_out_2" > "max_val" THEN
        "max_val" := "layer1_out_2";
    END_IF;
    IF "layer1_out_3" > "max_val" THEN
        "max_val" := "layer1_out_3";
    END_IF;
    IF "layer1_out_4" > "max_val" THEN
        "max_val" := "layer1_out_4";
    END_IF;
    "max_confidence" := "max_val";
    "predicted_class" := 1;
    IF "layer1_out_2" > "layer1_out_1" THEN
        "predicted_class" := 2;
    END_IF;
    IF "layer1_out_3" > "layer1_out_2" THEN
        "predicted_class" := 3;
    END_IF;
    IF "layer1_out_4" > "layer1_out_3" THEN
        "predicted_class" := 4;
    END_IF;
    "class_output_1" := "layer1_out_1";
    "class_output_2" := "layer1_out_2";
    "class_output_3" := "layer1_out_3";
    "class_output_4" := "layer1_out_4";

END_FUNCTION_BLOCK

// M2 bounds summary:
//   mean=0.8281
//   max=1.8567, M2*h^2/8(max)=0.04263
//   => de Boor bound satisfied: 0.04263 < 0.182